// TIA Portal V19 export
DATA_BLOCK "Config"   // DB68
// stored: MemoryReserve 100, Namespace Unit2
   VAR
      unit { ExternalWritable := 'False'} : "LAF_typeUnitConfiguration";   // Configuration of Unit Parameters
      stateMachine { ExternalWritable := 'False'} : "LUC_typeStateMachineConfiguration";
      signalStack { ExternalWritable := 'False'} : "LUC_typeSignalStackConfiguration";
      remoteCtrlOpcUa { ExternalWritable := 'False'} : "LUC_typeRemoteCtrlConfiguration";
      stateModeManager { ExternalAccessible := 'False'; ExternalVisible := 'False'; ExternalWritable := 'False'} : "LPMLV2022_typeConfiguration";   // Do not change. Can be configured through stateMachineConfiguration
      initConfigPar { S7_SetPoint := 'True'} : "UnitInitConfig";
   END_VAR
BEGIN
   unit.referenceDesignator.relative := WSTRING#'U1';
END_DATA_BLOCK
